// TIA Portal V19 export
TYPE "dtDrill"
   STRUCT
      level { S7_SetPoint := 'True'} : Array[0..3] of Int;
      tDelay { S7_SetPoint := 'True'} : Time := T#5s;
      setPriority { S7_SetPoint := 'True'} : Array[0..2] of Int;
      loadPriority : Array[0..2] of Int;
      TankAvailable : Array[0..1] of Bool;
      loadBtn : Bool;
   END_STRUCT;
   // level[0] := 80;
   // level[1] := 90;
   // level[2] := 95;
   // level[3] := 100;
   // setPriority[0..2] := 0;
END_TYPE
